Yaskawa INFORM job: X2_99(90,0).JBI

/JOB
//NAME X2_99(90,0)
///FOLDERNAME X2
//POS
///NPOS 429,429,425,13,0,0
///TOOL 0
///POSTYPE PULSE
///PULSE
C00000=-2065,-103387,-83817,35,52737,-27
C00001=166393,-132062,-92618,-58483,55149,-81008
C00002=157482,-99612,-82443,-50725,53832,76817
C00003=152781,-96239,-78741,-49340,50884,75750
C00004=150954,-94792,-77210,-48744,49760,75306
C00005=150957,-94045,-75225,-49281,49201,75681
C00006=151067,-94769,-77060,-48840,49767,75375
C00007=148896,-96259,-77631,-48213,48319,74911
C00008=154925,-106114,-81211,-52368,49780,77962
C00009=154976,-104737,-78409,-53070,49177,78455
C00010=153765,-101609,-77307,-52041,49068,77683
C00011=154727,-103781,-80113,-51957,49998,77663
C00012=157482,-99612,-82443,-50725,53832,76817
C00013=126812,-81448,-90767,-9472,77282,14340
C00014=120783,-85892,-98127,47,82159,-60
C00015=120791,-78998,-92147,45,82022,-58
C00016=120812,-59041,-81112,38,85486,-50
C00017=120812,-59638,-79752,38,84341,-50
C00018=120812,-59041,-81112,38,85486,-50
C00019=120792,-70899,-87175,45,83124,-57
C00020=120810,-72484,-85548,40,81307,-51
C00021=120817,-76009,-87202,37,80512,-50
C00022=120816,-72927,-85752,37,81205,-50
C00023=120792,-71723,-87920,45,83159,-57
C00024=120783,-85892,-98127,47,82159,-60
C00025=120841,-86418,-98444,30,82084,-41
C00026=120867,-62955,-84955,21,85839,-32
C00027=120862,-57449,-80347,23,85833,-34
C00028=120862,-58065,-78999,24,84687,-34
C00029=120862,-57449,-80347,23,85833,-34
C00030=120848,-76846,-90076,28,81853,-39
C00031=120700,-77430,-87681,72,80079,-89
C00032=120707,-73445,-85814,70,80978,-86
C00033=120700,-77430,-87681,72,80079,-89
C00034=120841,-86418,-98444,30,82084,-41
C00035=120877,-85820,-98106,19,82183,-30
C00036=120894,-60284,-82721,14,85837,-23
C00037=120891,-57831,-80469,15,85712,-24
C00038=120891,-58439,-79117,15,84567,-25
C00039=120891,-57831,-80469,15,85712,-24
C00040=120882,-76306,-89742,18,81925,-28
C00041=120632,-76849,-87581,92,80316,-111
C00042=120641,-72870,-85708,89,81208,-107
C00043=120899,-105607,-111704,13,80383,-24
C00044=120899,-105607,-111704,13,80383,-24
C00045=120329,-64675,-84682,181,84785,-205
C00046=120337,-61857,-81845,179,84488,-203
C00047=120337,-62228,-80870,179,83698,-204
C00048=120337,-61849,-81865,179,84506,-203
C00049=120308,-72964,-87409,188,82206,-216
C00050=112365,-66887,-81837,2540,82030,-2815
C00051=112466,-65041,-80903,2509,82400,-2777
C00052=112291,-68228,-82506,2565,81755,-2847
C00053=88690,-37051,-64863,22386,100281,-29037
C00054=90338,-32373,-60570,22143,99643,-28585
C00055=86677,-30127,-56933,28301,101078,-28609
C00056=87262,-30704,-57322,28229,100840,-28451
C00057=86036,-30845,-57417,28365,101220,-28810
C00058=80749,-50154,-73696,28906,103010,-30322
C00059=106026,-92840,-102541,4408,81700,-4909
C00060=104933,-21068,-63327,14588,98299,-15445
C00061=118026,-7058,-59426,-2478,121298,-42537
C00062=119206,-9959,-57512,-2402,118662,-42076
C00063=119679,-11008,-56668,-2374,117617,-41892
C00064=119678,-12040,-55711,-2348,116499,-41868
C00065=119679,-11008,-56668,-2374,117617,-41892
C00066=117888,-11929,-55575,-2351,116426,-42475
C00067=118578,-11982,-55616,-2350,116441,-42241
C00068=117888,-11929,-55575,-2351,116426,-42475
C00069=116239,-8118,-58416,-2447,120087,-43116
C00070=117941,-7017,-59404,-2478,121303,-42566
C00071=119121,-9922,-57492,-2402,118667,-42105
C00072=119594,-10972,-56650,-2375,117622,-41921
C00073=119593,-12004,-55694,-2348,116504,-41897
C00074=119594,-10972,-56650,-2375,117622,-41921
C00075=117972,-11968,-55595,-2351,116420,-42446
C00076=118663,-12020,-55635,-2349,116436,-42212
C00077=117972,-11968,-55595,-2351,116420,-42446
C00078=116323,-8162,-58441,-2447,120082,-43087
C00079=118213,-4464,-57342,-2479,121353,-42475
C00080=119375,-7335,-55445,-2404,118742,-42020
C00081=119840,-8375,-54609,-2376,117706,-41839
C00082=119839,-9401,-53662,-2350,116597,-41815
C00083=119840,-8375,-54609,-2376,117706,-41839
C00084=117787,-9255,-53494,-2353,116516,-42511
C00085=118466,-9310,-53537,-2352,116532,-42281
C00086=117787,-9255,-53494,-2353,116516,-42511
C00087=113921,-56504,-90793,659,90254,-43086
C00088=172997,-84117,-74043,-29270,60841,-12459
C00089=182497,-62439,-47217,-33561,35566,-5540
C00090=159932,16406,-23252,-17890,77970,-26070
C00091=160037,20332,-16581,-18068,76003,-25738
C00092=160078,21964,-13839,-18147,75202,-25602
C00093=160081,21492,-12606,-18227,74248,-25457
C00094=160088,21570,-12789,-18218,74396,-25476
C00095=160141,24413,-10063,-18259,74201,-25427
C00096=160088,21570,-12789,-18218,74396,-25476
C00097=159942,15886,-22293,-17945,77154,-25943
C00098=147845,25725,-14551,-15841,76328,-30554
C00099=147785,29164,-8153,-15217,74000,-30118
C00100=146391,29253,-6691,-12120,72163,-29888
C00101=146393,28810,-5449,-12184,71193,-29788
C00102=146383,28918,-5675,-12167,71382,-29809
C00103=146621,31717,-2885,-12295,71143,-29703
C00104=146383,28918,-5675,-12167,71382,-29809
C00105=147481,21483,-15847,-15359,72675,-30094
C00106=159281,-34086,-66545,-16207,79188,-23357
C00107=99248,-110920,-110752,20005,76383,-39509
C00108=66302,7791,-36486,37409,101463,8597
C00109=118447,29266,3056,46998,72230,30227
C00110=127168,50798,26938,44779,68662,26958
C00111=126741,52789,31626,47411,67245,26245
C00112=126739,52962,33479,47729,66520,25863
C00113=126722,52773,32881,47650,66716,25957
C00114=127164,55780,36224,47676,66131,25882
C00115=126722,52773,32881,47650,66716,25957
C00116=126349,45711,19766,44599,70372,27360
C00117=120505,26515,5919,45760,54508,48320
C00118=117448,33812,16008,47845,44948,58363
C00119=118470,38735,23995,49076,42786,57538
C00120=118868,40836,27368,49664,41907,57166
C00121=118868,41209,29429,50591,41201,56605
C00122=118874,41229,29076,50388,41345,56729
C00123=119426,43973,31977,50392,40796,56713
C00124=118874,41229,29076,50388,41345,56729
C00125=113429,42926,32106,63659,45667,52339
C00126=114748,48529,40817,65458,43685,51182
C00127=114893,50540,41231,64669,43936,51674
C00128=112305,42308,35228,66023,45399,50822
C00129=115273,50693,44169,66217,42928,50725
C00130=115426,53095,46610,68400,49137,42398
C00131=119344,57393,45281,61419,62909,27573
C00132=122643,57481,41003,55027,68134,22006
C00133=122245,55189,37420,54802,68977,22330
C00134=121107,49775,28783,54366,71151,23084
C00135=66302,7791,-36486,37409,101463,8597
C00136=87180,-51399,-85456,25144,96058,-16686
C00137=99248,-110920,-110752,20005,76383,-39509
C00138=111751,-62315,-95524,15437,88724,-33512
C00139=159281,-34086,-66545,-16207,79188,-23357
C00140=168180,19564,-18932,-27022,75314,-21681
C00141=167557,25730,-9148,-27095,72571,-21254
C00142=169085,37421,-2781,-29202,81184,-22287
C00143=169685,28444,-11845,-29359,82224,-22336
C00144=167557,25730,-9148,-27095,72571,-21254
C00145=149649,39094,-686,-15861,76123,-27675
C00146=150907,26639,-9385,-19166,68714,-26529
C00147=150787,22066,-16509,-18873,70615,-26886
C00148=159281,-34086,-66545,-16207,79188,-23357
C00149=152303,-102933,-107906,365,71882,-21471
C00150=121799,-34443,-59064,1710,93632,-36707
C00151=118945,163,-15392,1659,93503,-40633
C00152=120696,28796,14633,1549,89703,-40093
C00153=120597,41866,29081,1551,94027,-40072
C00154=120652,45714,33392,1563,96828,-40019
C00155=120580,21627,9250,1574,100354,-40001
C00156=120617,1336,-9032,1541,99246,-41820
C00157=120512,926,-9516,1535,99334,-41857
C00158=120163,-1908,-13337,1516,100237,-41964
C00159=118931,-1420,-16721,1449,102592,-42361
C00160=118945,163,-15392,1659,93503,-40633
C00161=120171,930,-10959,1582,91145,-40250
C00162=120660,1326,-9108,1553,90200,-40098
C00163=120694,25865,13192,1550,89085,-40100
C00164=120696,29026,16285,1550,88805,-40104
C00165=120258,23290,9189,1576,90234,-40233
C00166=119165,22386,4533,1644,92655,-40570
C00167=119181,24192,6266,1459,101602,-42286
C00168=120260,23811,9690,1517,99280,-41943
C00169=120693,23749,11149,1541,98342,-41806
C00170=120660,1326,-9108,1544,99287,-41805
C00171=120174,1432,-10536,1517,100229,-41961
C00172=118965,1918,-13913,1451,102579,-42349
C00173=119164,21752,3941,1459,101779,-42290
C00174=120255,21351,7351,1518,99456,-41942
C00175=120694,21281,8802,1542,98518,-41803
C00176=120641,1282,-9371,1543,99426,-41811
C00177=120163,-1908,-13337,1516,100237,-41964
C00178=118931,-1420,-16721,1449,102592,-42361
C00179=109578,15420,-7310,28367,110236,41857
C00180=109763,14188,-4345,27924,107995,41350
C00181=110205,13439,-3187,27787,106873,41241
C00182=131058,12711,-3863,29133,99851,47652
C00183=122151,9951,8068,53530,92588,44188
C00184=120623,10562,7326,53535,93941,44154
C00185=119164,10594,3761,53715,96134,44669
C00186=115308,-32515,-29810,53374,97452,43308
C00187=161838,-55085,-61541,-4908,86946,11244
C00188=151264,19092,-3987,-26397,112513,-34927
C00189=144058,12336,-10204,-27380,110553,-37342
C00190=143876,11528,-6807,-26938,108253,-36840
C00191=143883,12398,-4144,-26739,107186,-36580
C00192=138876,8905,-7310,-27290,105714,-38195
C00193=141808,11001,6672,-48404,103196,-38053
C00194=146391,20880,29557,-62395,105787,-26226
C00195=143524,10867,7651,-51737,104094,-37857
C00196=145724,13401,6310,-52003,106686,-38162
C00197=151264,19092,-3987,-26397,112513,-34927
C00198=161838,-55085,-61541,-4908,86946,11244
C00199=148116,-52831,-56464,-50581,83749,-77178
C00200=143654,-45216,-49088,-49944,80892,-77944
C00201=142056,-46762,-48840,-49795,79395,-77968
C00202=142218,-45304,-47887,-49802,79593,-77989
C00203=141353,-40392,-44909,-49565,79578,-78427
C00204=143095,-64861,-43193,-72743,55101,-56913
C00205=145645,-63649,-42384,-72835,56889,-56645
C00206=146567,-66336,-44709,-72863,57538,-56558
C00207=148638,-70217,-49243,-72528,59219,-56701
C00208=152439,-71702,-66380,-51300,83828,-74957
C00209=84213,-62636,-84550,16381,94117,-81885
C00210=95245,-30826,-59151,14149,92862,-78402
C00211=97191,-43170,-61473,15355,82699,-78714
C00212=98481,-44184,-62246,14992,82421,-78309
C00213=94037,-41035,-61513,16198,84364,-79567
C00214=63521,1839,6360,71273,102323,-80160
C00215=65526,-1458,4791,71319,100695,-80245
C00216=65441,-828,6596,71139,100483,-80605
C00217=61873,133,7709,70638,102845,-81131
C00218=97631,-84017,-82277,6042,71977,-80454
C00219=97631,-84017,-82277,6042,71977,-13540
C00220=100992,-100869,-74320,15072,37892,-15545
C00221=103157,-95187,-70426,13089,38023,-14317
C00222=103157,-92961,-65713,13621,36312,-14617
C00223=97699,-120955,-80408,20799,32327,-18909
C00224=-2043,-48212,-53796,8,82315,-15
C00225=-2043,-48212,-53796,8,82315,-15
C00226=-2043,-48212,-53796,8,82315,-15
C00227=-2043,-48212,-53796,8,82315,-15
C00228=-2043,-48212,-53796,8,82315,-15
C00229=50156,-143124,-107249,60088,69694,-78596
C00230=70410,-104162,-83449,55661,60383,-81011
C00231=84923,-92751,-76765,50721,53081,-76684
C00232=86734,-91468,-75289,50215,51915,-76295
C00233=86736,-90744,-73307,50726,51361,-76670
C00234=86623,-91438,-75136,50303,51925,-76361
C00235=88689,-93063,-75778,49797,50498,-75974
C00236=86623,-91438,-75136,50303,51925,-76361
C00237=82499,-102310,-79219,53526,52313,-78845
C00238=82460,-100986,-76424,54186,51705,-79335
C00239=83746,-97994,-75341,53258,51491,-78599
C00240=82460,-100986,-76424,54186,51705,-79335
C00241=83820,-89231,-90898,31984,73153,-45470
C00242=103333,-81093,-95821,5106,83352,-5547
C00243=105734,-58391,-81894,4383,86302,-4664
C00244=106051,-55558,-79074,4290,86007,-4572
C00245=106052,-56155,-77720,4294,84870,-4611
C00246=106051,-55558,-79074,4290,86007,-4572
C00247=104417,-72181,-87594,4790,82806,-5215
C00248=104401,-72744,-85473,4810,81218,-5281
C00249=104801,-68935,-83629,4684,82015,-5119
C00250=104401,-72744,-85473,4810,81218,-5281
C00251=103333,-81093,-95821,5106,83352,-5547
C00252=121034,-86160,-98106,-184,81635,191
C00253=120937,-60313,-84022,-154,86250,153
C00254=120931,-57182,-80055,-152,85416,152
C00255=120931,-57770,-78693,-152,84276,154
C00256=120931,-57182,-80055,-152,85416,152
C00257=120995,-76536,-89732,-172,81427,178
C00258=121142,-77068,-87314,-217,79666,229
C00259=121124,-73096,-85459,-211,80565,222
C00260=121142,-77068,-87314,-217,79666,229
C00261=121096,-115670,-111851,-205,74930,222
C00262=121096,-115670,-111851,-205,74930,222
C00263=111920,-77360,-89293,2569,80863,-2809
C00264=113418,-69208,-82911,2118,81083,-2310
C00265=113298,-70113,-82134,2157,80142,-2365
C00266=113298,-69851,-83365,2151,81033,-2349
C00267=112830,-79068,-87705,2304,78982,-2541
C00268=118405,-74923,-83336,614,78322,-682
C00269=118432,-73250,-82545,605,78695,-671
C00270=118359,-77891,-84712,629,77644,-701
C00271=147649,-49700,-70143,-21952,96038,28312
C00272=144092,-44169,-65180,-21423,94945,27268
C00273=143301,-44665,-65479,-21298,94683,27039
C00274=145130,-43494,-64769,-21581,95292,27566
C00275=153783,-86392,-93366,-22522,93398,30972
C00276=150910,-93017,-97560,-17688,85250,21630
C00277=120908,-62091,-84868,-144,85857,144
C00278=120903,-58004,-80414,-143,85215,144
C00279=120903,-58580,-79044,-143,84076,145
C00280=120903,-58004,-80414,-143,85215,144
C00281=120961,-76486,-89626,-161,81387,167
C00282=121210,-76970,-87437,-238,79792,251
C00283=121190,-72994,-85579,-231,80691,243
C00284=121210,-76970,-87437,-238,79792,251
C00285=120997,-86105,-97999,-172,81597,178
C00286=122173,-44832,-80249,1138,103105,21360
C00287=123342,-6609,-59067,2432,120936,42504
C00288=122164,-9458,-57119,2365,118305,42047
C00289=121693,-10486,-56262,2341,117263,41864
C00290=121692,-11496,-55292,2315,116147,41841
C00291=121693,-10486,-56262,2341,117263,41864
C00292=123082,-11418,-55178,2309,116084,42311
C00293=122789,-11440,-55197,2311,116090,42211
C00294=123477,-11388,-55156,2308,116075,42444
C00295=125124,-7649,-58044,2392,119728,43080
C00296=123427,-6569,-59045,2432,120941,42533
C00297=122249,-10161,-56477,2346,117547,42058
C00298=121777,-10451,-56245,2341,117268,41893
C00299=121777,-11461,-55275,2315,116153,41870
C00300=121777,-10451,-56245,2341,117268,41893
C00301=123393,-11428,-55177,2309,116069,42415
C00302=122704,-11478,-55216,2311,116085,42182
C00303=123393,-11428,-55177,2309,116069,42415
C00304=123141,-2998,-56146,2434,120999,42438
C00305=121991,-6366,-54527,2366,118305,41988
C00306=121527,-6824,-53376,2344,117373,41811
C00307=121527,-7826,-52419,2319,116269,41787
C00308=121527,-6824,-53376,2344,117373,41811
C00309=123560,-7684,-52253,2311,116189,42474
C00310=122887,-7737,-52295,2313,116204,42247
C00311=123560,-7684,-52253,2311,116189,42474
C00312=125171,-3981,-55094,2393,119797,43097
C00313=101327,-45531,-60072,2075,102128,34667
C00314=89266,4396,-33928,11465,93507,29927
C00315=71071,57081,18578,22711,75509,22099
C00316=71211,62019,27131,22931,72950,21646
C00317=71266,64149,30755,23040,71886,21453
C00318=71267,63961,32200,23162,70975,21270
C00319=71260,64000,31991,23145,71114,21296
C00320=71334,67369,35901,23203,70471,21193
C00321=71260,64000,31991,23145,71114,21296
C00322=71066,56762,19636,22790,74756,21949
C00323=94467,40678,813,12417,73109,29814
C00324=94083,44902,8245,12754,70817,29441
C00325=93934,46692,11343,12898,69876,29287
C00326=93935,46363,12659,12975,68921,29182
C00327=93944,46449,12421,12955,69106,29206
C00328=93737,49413,15622,13089,68702,29088
C00329=93944,46449,12421,12955,69106,29206
C00330=94477,40302,1770,12461,72343,29738
C00331=89266,4396,-33928,11465,93507,29927
C00332=101327,-45531,-60072,2075,102128,34667
C00333=154347,-58865,-59313,-31959,84488,-20300
C00334=132804,-7309,-34611,-38234,83249,-26564
C00335=122176,70455,38125,-50476,77977,-25755
C00336=115295,79862,53015,-49496,71409,-25751
C00337=115674,81709,55615,-49754,71183,-25426
C00338=115674,81913,57390,-49999,70533,-25064
C00339=115723,81771,56361,-49871,70928,-25259
C00340=115127,86395,62081,-50016,69849,-24976
C00341=115723,81734,56059,-49831,71039,-25319
C00342=117859,70375,39301,-49439,75156,-26443
C00343=124576,6255,-12780,-47438,56902,-47453
C00344=122250,19334,1935,-46182,44641,-59320
C00345=122250,19334,1935,-46182,44641,-59320
C00346=120782,25934,12333,-47564,41782,-58376
C00347=120782,26215,14271,-48443,41066,-57848
C00348=120776,26249,13930,-48246,41217,-57966
C00349=120208,28831,16455,-48074,40759,-58046
C00350=120776,26249,13930,-48246,41217,-57966
C00351=118681,43368,36578,-62815,38306,-52785
C00352=118657,41916,32618,-60942,39123,-53866
C00353=119090,39280,31915,-62143,38937,-53171
C00354=118568,43405,36686,-62818,38211,-52783
C00355=112564,55763,35688,-55377,68087,-24843
C00356=113391,48910,28472,-52811,66916,-24378
C00357=112985,43681,22401,-52223,67232,-24845
C00358=132804,-7309,-34611,-38234,83249,-26564
C00359=154347,-58865,-59313,-31959,84488,-20300
C00360=101327,-45531,-60072,2075,102128,34667
C00361=89266,4396,-33928,11465,93507,29927
C00362=66565,54061,16600,30569,73521,18779
C00363=67024,59337,25188,30775,71132,18293
C00364=67157,61403,28617,30898,70179,18077
C00365=81564,59654,26436,24505,65914,22675
C00366=81641,57287,22841,24296,66807,22900
C00367=81527,51927,14208,23948,69183,23371
C00368=78027,-14448,-47618,10307,89336,23924
C00369=122403,540,-15029,-1679,93098,40614
C00370=116416,39963,24023,-1992,100377,38466
C00371=113398,50152,38563,-2230,96586,37494
C00372=112489,24468,12107,-2384,100085,37116
C00373=111594,3062,-7595,-2103,98667,38669
C00374=111355,667,-9500,-2114,98597,38588
C00375=111941,198,-11543,-2089,99632,38773
C00376=113186,289,-15256,-2035,101994,39161
C00377=122403,540,-15029,-1679,93098,40614
C00378=121179,1356,-10556,-1597,90741,40233
C00379=120574,1774,-8687,-1557,89793,40041
C00380=120532,26429,13697,-1554,88684,40039
C00381=121099,23723,9564,-1591,89850,40218
C00382=122190,22771,4863,-1663,92275,40553
C00383=122175,24579,6594,-1485,101224,42269
C00384=121098,24245,10065,-1538,98897,41927
C00385=120630,24202,11544,-1561,97957,41779
C00386=120666,1773,-8688,-1564,98883,41779
C00387=121177,1858,-10134,-1538,99825,41943
C00388=122384,2295,-13553,-1478,102176,42330
C00389=122189,22661,4761,-1485,101367,42272
C00390=121101,22312,8220,-1538,99039,41927
C00391=120664,22262,9692,-1560,98100,41789
C00392=120644,766,-9415,-1564,98810,41771
C00393=121185,-971,-12517,-1537,99838,41946
C00394=122412,-533,-15942,-1476,102193,42339
C00395=131781,15460,-7279,-28376,109886,-41795
C00396=131592,14275,-4268,-27940,107640,-41290
C00397=130646,14147,-2566,-27857,106338,-41338
C00398=110382,14201,-2350,-29042,99390,-47524
C00399=119227,11935,9973,-53508,92244,-44000
C00400=120732,10849,7590,-53521,93669,-44023
C00401=122191,10834,3980,-53696,95864,-44539
C00402=128646,-26020,-30624,-53883,101032,-13133
C00403=66557,-34885,-48546,20214,102394,2504
C00404=79484,36547,13079,24373,114005,30975
C00405=85904,26694,3247,25718,112997,33343
C00406=86041,25965,6661,25253,110710,32858
C00407=85714,26763,9282,24984,109715,32500
C00408=90422,20837,3523,25806,108738,34143
C00409=87739,24554,20424,48221,108657,34815
C00410=84755,20942,20954,53722,106133,35573
C00411=84755,20942,20954,53722,106133,35573
C00412=84776,24179,21069,50511,109377,34699
C00413=84698,26318,18454,50015,112057,35133
C00414=81578,31234,5255,15438,110633,30982
C00415=71416,-31459,-49219,37385,106309,54903
C00416=79334,-27512,-40554,52438,93314,75230
C00417=81671,-29746,-39165,52092,90747,74997
C00418=82501,-31675,-39268,51984,89697,74838
C00419=82828,-30755,-38544,51956,89529,74918
C00420=84142,-26044,-35343,51821,89078,75358
C00421=80223,-43644,-36659,65279,74230,62526
C00422=80042,-45349,-41066,60562,72331,65280
C00423=77493,-50941,-36554,72626,70323,55695
C00424=74018,-52299,-39928,72336,73171,55924
C00425=60945,-55409,-65093,53734,104166,71681
C00426=60945,-55409,-65093,53734,104166,71681
C00427=122092,-114409,-88723,-8345,70481,11232
C00428=-2000,-48025,-60869,0,102856,0
BC00000=781,523905,302382
BC00001=30742,515701,66855
BC00002=31638,515479,60490
BC00003=31638,515479,60490
BC00004=31638,515479,60490
BC00005=31638,515479,60490
BC00006=31638,515479,60490
BC00007=31638,515479,60490
BC00008=31638,515479,60490
BC00009=31638,515479,60490
BC00010=31638,515479,60490
BC00011=31638,515479,60490
BC00012=31638,515479,60490
BC00013=13239,522628,91328
BC00014=10409,517207,59294
BC00015=10409,517207,59294
BC00016=10409,517207,59294
BC00017=10409,517207,59294
BC00018=10409,517207,59294
BC00019=10409,517207,59294
BC00020=10409,517207,59294
BC00021=10409,517207,59294
BC00022=10409,517207,59294
BC00023=10409,517207,59294
BC00024=10409,517207,59294
BC00025=68218,516454,58706
BC00026=68218,516454,58706
BC00027=68218,516454,58706
BC00028=68218,516454,58706
BC00029=68218,516454,58706
BC00030=68218,516454,58706
BC00031=68218,516454,58706
BC00032=68218,516454,58706
BC00033=68218,516454,58706
BC00034=68218,516454,58706
BC00035=126843,516488,59263
BC00036=126843,516488,59263
BC00037=126843,516488,59263
BC00038=126843,516488,59263
BC00039=126843,516488,59263
BC00040=126843,516488,59263
BC00041=126843,516488,59263
BC00042=126843,516488,59263
BC00043=126843,520400,59263
BC00044=387083,520400,59263
BC00045=387083,520400,59263
BC00046=387083,520400,59263
BC00047=387083,520400,59263
BC00048=387083,520400,59263
BC00049=387083,520400,59263
BC00050=387083,520400,59263
BC00051=387083,520400,59263
BC00052=387083,520400,59263
BC00053=387083,520400,59263
BC00054=387083,520400,59263
BC00055=387083,520400,59263
BC00056=387083,520400,59263
BC00057=387083,520400,59263
BC00058=387083,520400,59263
BC00059=126843,518210,59263
BC00060=126843,518210,59263
BC00061=129574,490644,58205
BC00062=129574,490644,58205
BC00063=129574,490644,58205
BC00064=129574,490644,58205
BC00065=129574,490644,58205
BC00066=129574,490644,58205
BC00067=129574,490644,58205
BC00068=129574,490644,58205
BC00069=129574,490644,58205
BC00070=129597,444075,57932
BC00071=129597,444075,57932
BC00072=129597,444075,57932
BC00073=129597,444075,57932
BC00074=129597,444075,57932
BC00075=129597,444075,57932
BC00076=129597,444075,57932
BC00077=129597,444075,57932
BC00078=129597,444075,57932
BC00079=128889,400556,57777
BC00080=128889,400556,57777
BC00081=128889,400556,57777
BC00082=128889,400556,57777
BC00083=128889,400556,57777
BC00084=128889,400556,57777
BC00085=128889,400556,57777
BC00086=128889,400556,57777
BC00087=128889,400556,57777
BC00088=181249,400556,192761
BC00089=202914,400556,241573
BC00090=123650,400556,63155
BC00091=123650,400556,63155
BC00092=123650,400556,63155
BC00093=123650,400556,63155
BC00094=123650,400556,63155
BC00095=123650,400556,63155
BC00096=123650,400556,63155
BC00097=123650,400556,63155
BC00098=128418,400556,63301
BC00099=128418,400556,63301
BC00100=128418,400556,63301
BC00101=128418,400556,63301
BC00102=128418,400556,63301
BC00103=128418,400556,63301
BC00104=128418,400556,63301
BC00105=128418,400556,63301
BC00106=120912,400556,90455
BC00107=91224,400556,32086
BC00108=60523,400556,81483
BC00109=120036,400556,87759
BC00110=141181,415917,88489
BC00111=141181,415917,88489
BC00112=141181,415917,88489
BC00113=141181,415917,88489
BC00114=141181,415917,88489
BC00115=141181,415917,88489
BC00116=141181,415917,88489
BC00117=135777,415917,84971
BC00118=132933,415917,83120
BC00119=132933,415917,83120
BC00120=132933,415917,83120
BC00121=132933,415917,83120
BC00122=132933,415917,83120
BC00123=132933,415917,83120
BC00124=132933,415917,83120
BC00125=133247,415917,81483
BC00126=133247,415917,81483
BC00127=133247,415917,81483
BC00128=133247,415917,81483
BC00129=133246,415917,81483
BC00130=133247,415917,81482
BC00131=133247,415917,81483
BC00132=133247,415917,81483
BC00133=133247,415917,81483
BC00134=133247,415917,81483
BC00135=60523,400556,81483
BC00136=78278,400556,52915
BC00137=91224,400556,32086
BC00138=91224,400556,32086
BC00139=120912,400556,90455
BC00140=136017,400556,32086
BC00141=136017,400556,32086
BC00142=136017,400556,32086
BC00143=136017,400556,32086
BC00144=136017,400556,32086
BC00145=136017,400556,32086
BC00146=136017,400556,32086
BC00147=136017,400556,32086
BC00148=120912,400556,90455
BC00149=158121,400556,32086
BC00150=123507,424612,191697
BC00151=141020,441223,281235
BC00152=141020,441223,281235
BC00153=141020,441223,281235
BC00154=141020,441223,281235
BC00155=141020,441223,281235
BC00156=141154,470147,281572
BC00157=141330,514662,281853
BC00158=141330,514662,281853
BC00159=141330,514662,281853
BC00160=143409,441223,281235
BC00161=143409,441223,281235
BC00162=143409,441223,281235
BC00163=143409,441223,281235
BC00164=143409,441223,281235
BC00165=143409,441223,281235
BC00166=143409,441223,281235
BC00167=143543,470147,281572
BC00168=143543,470147,281572
BC00169=143543,470147,281572
BC00170=143543,470147,281572
BC00171=143543,470147,281572
BC00172=143543,470147,281572
BC00173=143719,514662,281853
BC00174=143719,514662,281853
BC00175=143719,514662,281853
BC00176=143719,514662,281853
BC00177=143719,514662,281853
BC00178=143719,514662,281853
BC00179=144290,523889,221847
BC00180=144290,523889,221847
BC00181=144290,523889,221847
BC00182=144290,523889,221847
BC00183=144290,523889,221845
BC00184=144290,523889,221847
BC00185=144290,523889,221847
BC00186=144290,523889,221847
BC00187=796,523889,224399
BC00188=796,523889,224399
BC00189=796,523889,224399
BC00190=796,523889,224399
BC00191=796,523889,224399
BC00192=796,523889,224399
BC00193=796,523889,224399
BC00194=796,523889,224399
BC00195=796,523889,224399
BC00196=796,523889,224399
BC00197=796,523889,224399
BC00198=796,523889,224399
BC00199=797,523888,121430
BC00200=796,523889,121434
BC00201=796,523889,121434
BC00202=796,523889,121434
BC00203=796,523889,121434
BC00204=796,523889,121434
BC00205=796,523889,121434
BC00206=796,523889,121434
BC00207=796,523889,121434
BC00208=796,523889,121434
BC00209=380682,523889,121434
BC00210=380682,523889,121434
BC00211=380682,523889,121434
BC00212=380682,523889,121434
BC00213=380682,523889,121434
BC00214=380682,523889,121434
BC00215=380682,523889,121434
BC00216=380682,523889,121434
BC00217=380682,523889,121434
BC00218=380682,523889,121434
BC00219=380682,523889,121434
BC00220=380682,523889,121434
BC00221=380682,523889,121434
BC00222=380682,523889,121434
BC00223=380682,523889,121434
BC00224=796,523889,1075193
BC00225=796,523889,1075193
BC00226=796,523889,1075193
BC00227=796,523889,1075193
BC00228=796,584159,1075193
BC00229=395769,514369,57931
BC00230=395769,514369,57931
BC00231=395769,514369,57931
BC00232=395769,514369,57931
BC00233=395769,514369,57931
BC00234=395769,514369,57931
BC00235=395769,514369,57931
BC00236=395769,514369,57931
BC00237=395769,514369,57931
BC00238=395769,514369,57931
BC00239=395769,514369,57931
BC00240=395769,514369,57931
BC00241=395769,515177,57354
BC00242=395769,516086,56705
BC00243=395769,516086,56705
BC00244=395769,516086,56705
BC00245=395769,516086,56705
BC00246=395769,516086,56705
BC00247=395769,516086,56705
BC00248=395769,516086,56705
BC00249=395769,516086,56705
BC00250=395769,516086,56705
BC00251=395769,516086,56705
BC00252=364519,515355,56108
BC00253=364519,515355,56108
BC00254=364519,515355,56108
BC00255=364519,515355,56108
BC00256=364519,515355,56108
BC00257=364519,515355,56108
BC00258=364519,515355,56108
BC00259=364519,515355,56108
BC00260=364519,515355,56108
BC00261=364519,515355,56108
BC00262=28307,515355,56108
BC00263=28307,516891,68607
BC00264=28307,516891,73984
BC00265=28307,516891,73984
BC00266=28307,516891,73984
BC00267=28307,516891,73984
BC00268=28307,516891,73984
BC00269=28307,516891,73984
BC00270=28307,516891,73984
BC00271=28307,516891,73984
BC00272=28307,516891,73984
BC00273=28307,516891,73984
BC00274=28307,516891,73984
BC00275=28307,516891,73984
BC00276=336711,509467,91104
BC00277=305893,515413,56636
BC00278=305893,515413,56636
BC00279=305893,515413,56636
BC00280=305893,515413,56636
BC00281=305893,515413,56636
BC00282=305893,515413,56636
BC00283=305893,515413,56636
BC00284=305893,515413,56636
BC00285=305893,515413,56636
BC00286=304523,502491,56408
BC00287=303152,489569,56181
BC00288=303152,489569,56181
BC00289=303152,489569,56181
BC00290=303152,489569,56181
BC00291=303152,489569,56181
BC00292=303152,489569,56181
BC00293=303152,489569,56181
BC00294=303152,489569,56181
BC00295=303152,489569,56181
BC00296=303109,443000,56994
BC00297=303109,443000,56994
BC00298=303109,443000,56994
BC00299=303109,443000,56994
BC00300=303109,443000,56994
BC00301=303109,443000,56994
BC00302=303109,443000,56994
BC00303=303109,443000,56994
BC00304=303797,400556,57919
BC00305=303797,400556,57919
BC00306=303797,400556,57919
BC00307=303797,400556,57919
BC00308=303797,400556,57919
BC00309=303797,400556,57919
BC00310=303797,400556,57919
BC00311=303797,400556,57919
BC00312=303797,400556,57919
BC00313=303797,400556,221955
BC00314=296099,410471,136295
BC00315=257856,418698,65216
BC00316=257856,418698,65216
BC00317=257856,418698,65216
BC00318=257856,418698,65216
BC00319=257856,418698,65216
BC00320=257856,418698,65216
BC00321=257856,418698,65216
BC00322=257856,418698,65216
BC00323=294733,415445,65881
BC00324=294733,415445,65881
BC00325=294733,415445,65881
BC00326=294733,415445,65881
BC00327=294733,415445,65881
BC00328=294733,415445,65881
BC00329=294733,415445,65881
BC00330=294733,415445,65881
BC00331=296099,410471,136295
BC00332=303797,400556,221955
BC00333=303797,400556,221955
BC00334=298676,400556,147304
BC00335=307528,431278,26398
BC00336=283636,431278,26398
BC00337=283636,431278,26398
BC00338=283636,431278,26398
BC00339=283636,431278,26398
BC00340=283636,431278,26398
BC00341=283636,431278,26398
BC00342=283636,431278,26398
BC00343=294823,400556,85625
BC00344=294931,400556,84298
BC00345=294931,400556,84298
BC00346=294931,400556,84298
BC00347=294931,400556,84298
BC00348=294931,400556,84298
BC00349=294931,400556,84298
BC00350=294931,400556,84298
BC00351=276015,408236,82027
BC00352=276015,408236,82027
BC00353=276015,408236,82027
BC00354=276015,408236,82027
BC00355=275463,408352,55361
BC00356=276012,408236,82027
BC00357=276015,408236,82027
BC00358=298676,400556,147304
BC00359=303797,400556,221955
BC00360=303797,400556,221955
BC00361=296099,410471,136295
BC00362=257149,416120,34454
BC00363=257149,416120,34454
BC00364=257149,416120,34454
BC00365=257149,416120,34454
BC00366=257149,416120,34454
BC00367=257149,416120,34454
BC00368=262502,428258,159266
BC00369=291631,440131,281365
BC00370=278652,440131,281365
BC00371=267739,440131,281365
BC00372=267739,440131,281365
BC00373=267671,469055,280615
BC00374=267515,514115,279786
BC00375=267515,514115,279786
BC00376=267515,514115,279786
BC00377=294020,440131,281365
BC00378=294020,440131,281365
BC00379=294020,440131,281365
BC00380=294020,440131,281365
BC00381=294020,440131,281365
BC00382=294020,440131,281365
BC00383=293952,469055,280615
BC00384=293952,469055,280615
BC00385=293952,469055,280615
BC00386=293952,469055,280615
BC00387=293952,469055,280615
BC00388=293952,469055,280615
BC00389=293796,514115,279786
BC00390=293796,514115,279786
BC00391=293796,514115,279786
BC00392=293796,514115,279786
BC00393=293796,514115,279786
BC00394=293796,514115,279786
BC00395=288422,523889,220135
BC00396=288422,523889,220135
BC00397=288422,523889,220135
BC00398=288422,523889,220135
BC00399=288422,523889,220135
BC00400=288422,523889,220135
BC00401=288422,523889,220135
BC00402=288422,523889,220135
BC00403=395769,523889,222081
BC00404=395769,523889,222081
BC00405=395769,523889,222081
BC00406=395769,523889,222081
BC00407=395769,523889,222081
BC00408=395769,523889,222081
BC00409=395769,523889,222080
BC00410=395769,523889,222080
BC00411=395769,523889,222080
BC00412=395769,523889,222081
BC00413=395769,523889,222081
BC00414=395769,523889,222081
BC00415=395769,523889,160664
BC00416=395769,523889,116189
BC00417=395769,523889,116189
BC00418=395769,523889,116189
BC00419=395769,523889,116189
BC00420=395769,523889,116189
BC00421=395769,523889,116189
BC00422=395769,523889,116189
BC00423=395769,523889,116189
BC00424=395769,523889,116189
BC00425=395769,523889,116189
BC00426=56749,523889,116189
BC00427=63741,523891,182530
BC00428=116059,523905,678960
EC00000=-798156,-183832
EC00001=-798156,-183832
EC00002=-798156,-183832
EC00003=-798156,-183832
EC00004=-798156,-183832
EC00005=-798156,-183832
EC00006=-798156,-183832
EC00007=-798156,-183832
EC00008=-798156,-183832
EC00009=-798156,-183832
EC00010=-798156,-183832
EC00011=-798156,-183832
EC00012=-798156,-183832
EC00013=-798156,-183832
EC00014=-798156,-183832
EC00015=-798156,-183832
EC00016=-798156,-183832
EC00017=-798156,-183832
EC00018=-798156,-183832
EC00019=-798156,-183832
EC00020=-798156,-183832
EC00021=-798156,-183832
EC00022=-798156,-183832
EC00023=-798156,-183832
EC00024=-798156,-183832
EC00025=-798156,-183832
EC00026=-798156,-183832
EC00027=-798156,-183832
EC00028=-798156,-183832
EC00029=-798156,-183832
EC00030=-798156,-183832
EC00031=-798156,-183832
EC00032=-798156,-183832
EC00033=-798156,-183832
EC00034=-798156,-183832
EC00035=-798156,-183832
EC00036=-798156,-183832
EC00037=-798156,-183832
EC00038=-798156,-183832
EC00039=-798156,-183832
EC00040=-798156,-183832
EC00041=-798156,-183832
EC00042=-798156,-183832
EC00043=-798156,-183832
EC00044=-798156,-183832
EC00045=-798156,-183832
EC00046=-798156,-183832
EC00047=-798156,-183832
EC00048=-798156,-183832
EC00049=-798156,-183832
EC00050=-798156,-183832
EC00051=-798156,-183832
EC00052=-798156,-183832
EC00053=-798156,-183832
EC00054=-798156,-183832
EC00055=-798156,-183832
EC00056=-798156,-183832
EC00057=-798156,-183832
EC00058=-798156,-183832
EC00059=-798156,-183832
EC00060=-798156,-183832
EC00061=-798156,-183832
EC00062=-798156,-183832
EC00063=-798156,-183832
EC00064=-798156,-183832
EC00065=-798156,-183832
EC00066=-798156,-183832
EC00067=-798156,-183832
EC00068=-798156,-183832
EC00069=-798156,-183832
EC00070=-798156,-183832
EC00071=-798156,-183832
EC00072=-798156,-183832
EC00073=-798156,-183832
EC00074=-798156,-183832
EC00075=-798156,-183832
EC00076=-798156,-183832
EC00077=-798156,-183832
EC00078=-798156,-183832
EC00079=-798156,-183832
EC00080=-798156,-183832
EC00081=-798156,-183832
EC00082=-798156,-183832
EC00083=-798156,-183832
EC00084=-798156,-183832
EC00085=-798156,-183832
EC00086=-798156,-183832
EC00087=-798156,-183832
EC00088=-798156,-183832
EC00089=-798156,-183832
EC00090=-798156,-183832
EC00091=-798156,-183832
EC00092=-798156,-183832
EC00093=-798156,-183832
EC00094=-798156,-183832
EC00095=-798156,-183832
EC00096=-798156,-183832
EC00097=-798156,-183832
EC00098=-798156,-183832
EC00099=-798156,-183832
EC00100=-798156,-183832
EC00101=-798156,-183832
EC00102=-798156,-183832
EC00103=-798156,-183832
EC00104=-798156,-183832
EC00105=-798156,-183832
EC00106=-798156,-183832
EC00107=-798156,-183832
EC00108=-798156,-183832
EC00109=-798156,-183832
EC00110=-798156,-183832
EC00111=-798156,-183832
EC00112=-798156,-183832
EC00113=-798156,-183832
EC00114=-798156,-183832
EC00115=-798156,-183832
EC00116=-798156,-183832
EC00117=-798156,-183832
EC00118=-798156,-183832
EC00119=-798156,-183832
EC00120=-798156,-183832
EC00121=-798156,-183832
EC00122=-798156,-183832
EC00123=-798156,-183832
EC00124=-798156,-183832
EC00125=-798156,-183832
EC00126=-798156,-183832
EC00127=-798155,-183833
EC00128=-798155,-183833
EC00129=-798156,-183832
EC00130=-798156,-183832
EC00131=-798156,-183832
EC00132=-798156,-183832
EC00133=-798156,-183832
EC00134=-798156,-183832
EC00135=-798156,-183832
EC00136=-798156,-183832
EC00137=-798156,-183832
EC00138=-798156,-183832
EC00139=-798156,-183832
EC00140=-798156,-183832
EC00141=-798156,-183832
EC00142=-798156,-183832
EC00143=-798156,-183832
EC00144=-798156,-183832
EC00145=-798156,-183832
EC00146=-798156,-183832
EC00147=-798156,-183832
EC00148=-798156,-183832
EC00149=-798156,-183832
EC00150=-798156,-183832
EC00151=-798156,-183832
EC00152=-798156,-183832
EC00153=-798156,-183832
EC00154=-798156,-183832
EC00155=-798156,-183832
EC00156=-798156,-183832
EC00157=-798156,-183832
EC00158=-798156,-183832
EC00159=-798156,-183832
EC00160=-798156,-183832
EC00161=-798156,-183832
EC00162=-798156,-183832
EC00163=-798156,-183832
EC00164=-798156,-183832
EC00165=-798156,-183832
EC00166=-798156,-183832
EC00167=-798156,-183832
EC00168=-798156,-183832
EC00169=-798156,-183832
EC00170=-798156,-183832
EC00171=-798156,-183832
EC00172=-798156,-183832
EC00173=-798156,-183832
EC00174=-798156,-183832
EC00175=-798156,-183832
EC00176=-798156,-183832
EC00177=-798156,-183832
EC00178=-798156,-183832
EC00179=-798155,-183833
EC00180=-798156,-183832
EC00181=-798156,-183832
EC00182=-798156,-183832
EC00183=-798156,-183832
EC00184=-798156,-183832
EC00185=-798156,-183832
EC00186=-798156,-183832
EC00187=-798156,-183832
EC00188=-798156,-183832
EC00189=-798156,-183832
EC00190=-798156,-183832
EC00191=-798156,-183832
EC00192=-798156,-183832
EC00193=-798156,-183832
EC00194=-798156,-183832
EC00195=-798155,-183832
EC00196=-798156,-183832
EC00197=-798156,-183832
EC00198=-798156,-183832
EC00199=-798156,-183832
EC00200=-798156,-183832
EC00201=-798156,-183832
EC00202=-798156,-183832
EC00203=-798156,-183832
EC00204=-798156,-183832
EC00205=-798156,-183832
EC00206=-798156,-183832
EC00207=-798156,-183832
EC00208=-798156,-183832
EC00209=-798156,-183832
EC00210=-798156,-183832
EC00211=-798156,-183832
EC00212=-798156,-183832
EC00213=-798156,-183832
EC00214=-798156,-183832
EC00215=-798156,-183832
EC00216=-798156,-183832
EC00217=-798156,-183832
EC00218=-798156,-183832
EC00219=-798156,-183832
EC00220=-798156,-183832
EC00221=-310394,-183832
EC00222=-310394,-740307
EC00223=-310394,-1296783
EC00224=-798156,-1296783
EC00225=-798156,-1296783
EC00226=-798156,-1296783
EC00227=-798156,-1296783
EC00228=-798156,-1296783
EC00229=-798156,-1296783
EC00230=-798156,-1296783
EC00231=-798156,-1296783
EC00232=-798156,-1296783
EC00233=-798156,-1296783
EC00234=-798156,-1296783
EC00235=-798156,-1296783
EC00236=-798156,-1296783
EC00237=-798156,-1296783
EC00238=-798156,-1296783
EC00239=-798156,-1296783
EC00240=-798156,-1296783
EC00241=-798156,-1296783
EC00242=-798156,-1296783
EC00243=-798156,-1296783
EC00244=-798156,-1296783
EC00245=-798156,-1296783
EC00246=-798156,-1296783
EC00247=-798156,-1296783
EC00248=-798156,-1296783
EC00249=-798156,-1296783
EC00250=-798156,-1296783
EC00251=-798156,-1296783
EC00252=-798156,-1296783
EC00253=-798156,-1296783
EC00254=-798156,-1296783
EC00255=-798156,-1296783
EC00256=-798156,-1296783
EC00257=-798156,-1296783
EC00258=-798156,-1296783
EC00259=-798156,-1296783
EC00260=-798156,-1296783
EC00261=-798156,-1296783
EC00262=-798156,-1296783
EC00263=-798156,-1296783
EC00264=-798156,-1296783
EC00265=-798156,-1296783
EC00266=-798156,-1296783
EC00267=-798156,-1296783
EC00268=-798156,-1296783
EC00269=-798156,-1296783
EC00270=-798156,-1296783
EC00271=-798156,-1296783
EC00272=-798156,-1296783
EC00273=-798156,-1296783
EC00274=-798156,-1296783
EC00275=-798156,-1296783
EC00276=-798156,-1296783
EC00277=-798156,-1296783
EC00278=-798156,-1296783
EC00279=-798156,-1296783
EC00280=-798156,-1296783
EC00281=-798156,-1296783
EC00282=-798156,-1296783
EC00283=-798156,-1296783
EC00284=-798156,-1296783
EC00285=-798156,-1296783
EC00286=-798156,-1296783
EC00287=-798156,-1296783
EC00288=-798156,-1296783
EC00289=-798156,-1296783
EC00290=-798156,-1296783
EC00291=-798156,-1296783
EC00292=-798156,-1296783
EC00293=-798156,-1296783
EC00294=-798156,-1296783
EC00295=-798156,-1296783
EC00296=-798156,-1296783
EC00297=-798156,-1296783
EC00298=-798156,-1296783
EC00299=-798156,-1296783
EC00300=-798156,-1296783
EC00301=-798156,-1296783
EC00302=-798156,-1296783
EC00303=-798156,-1296783
EC00304=-798156,-1296783
EC00305=-798156,-1296783
EC00306=-798156,-1296783
EC00307=-798156,-1296783
EC00308=-798156,-1296783
EC00309=-798156,-1296783
EC00310=-798156,-1296783
EC00311=-798156,-1296783
EC00312=-798156,-1296783
EC00313=-798156,-1296783
EC00314=-798156,-1296783
EC00315=-798156,-1296783
EC00316=-798156,-1296783
EC00317=-798156,-1296783
EC00318=-798156,-1296783
EC00319=-798156,-1296783
EC00320=-798156,-1296783
EC00321=-798156,-1296783
EC00322=-798156,-1296783
EC00323=-798156,-1296783
EC00324=-798156,-1296783
EC00325=-798156,-1296783
EC00326=-798156,-1296783
EC00327=-798156,-1296783
EC00328=-798156,-1296783
EC00329=-798156,-1296783
EC00330=-798156,-1296783
EC00331=-798156,-1296783
EC00332=-798156,-1296783
EC00333=-798156,-1296783
EC00334=-798156,-1296783
EC00335=-798156,-1296783
EC00336=-798156,-1296783
EC00337=-798156,-1296783
EC00338=-798156,-1296783
EC00339=-798156,-1296783
EC00340=-798156,-1296783
EC00341=-798156,-1296783
EC00342=-798156,-1296783
EC00343=-798156,-1296783
EC00344=-798156,-1296783
EC00345=-798156,-1296783
EC00346=-798156,-1296783
EC00347=-798156,-1296783
EC00348=-798156,-1296783
EC00349=-798156,-1296783
EC00350=-798156,-1296783
EC00351=-798156,-1296783
EC00352=-798156,-1296783
EC00353=-798156,-1296783
EC00354=-798156,-1296783
EC00355=-798156,-1296783
EC00356=-798156,-1296783
EC00357=-798156,-1296783
EC00358=-798156,-1296783
EC00359=-798156,-1296783
EC00360=-798156,-1296783
EC00361=-798156,-1296783
EC00362=-798156,-1296783
EC00363=-798156,-1296783
EC00364=-798156,-1296783
EC00365=-798156,-1296783
EC00366=-798156,-1296783
EC00367=-798156,-1296783
EC00368=-798156,-1296783
EC00369=-798156,-1296783
EC00370=-798156,-1296783
EC00371=-798156,-1296783
EC00372=-798156,-1296783
EC00373=-798156,-1296783
EC00374=-798156,-1296783
EC00375=-798156,-1296783
EC00376=-798156,-1296783
EC00377=-798156,-1296783
EC00378=-798156,-1296783
EC00379=-798156,-1296783
EC00380=-798156,-1296783
EC00381=-798156,-1296783
EC00382=-798156,-1296783
EC00383=-798156,-1296783
EC00384=-798156,-1296783
EC00385=-798156,-1296783
EC00386=-798156,-1296783
EC00387=-798156,-1296783
EC00388=-798156,-1296783
EC00389=-798156,-1296783
EC00390=-798156,-1296783
EC00391=-798156,-1296783
EC00392=-798156,-1296783
EC00393=-798156,-1296783
EC00394=-798156,-1296783
EC00395=-798156,-1296783
EC00396=-798156,-1296783
EC00397=-798156,-1296783
EC00398=-798156,-1296783
EC00399=-798156,-1296783
EC00400=-798156,-1296783
EC00401=-798156,-1296783
EC00402=-798156,-1296783
EC00403=-798156,-1296783
EC00404=-798156,-1296783
EC00405=-798154,-1296781
EC00406=-798154,-1296781
EC00407=-798154,-1296781
EC00408=-798155,-1296782
EC00409=-798156,-1296783
EC00410=-798156,-1296783
EC00411=-798156,-1296783
EC00412=-798156,-1296783
EC00413=-798156,-1296783
EC00414=-798156,-1296783
EC00415=-798156,-1296783
EC00416=-798156,-1296783
EC00417=-798156,-1296783
EC00418=-798156,-1296783
EC00419=-798156,-1296783
EC00420=-798156,-1296783
EC00421=-798156,-1296783
EC00422=-798156,-1296783
EC00423=-798154,-1296780
EC00424=-798156,-1296783
///POSTYPE BASE
///RECTAN
///RCONF 0,0,0,0,1,0,0,0,0,0,0,0,0,0,0,0,0,0,0,0,0,0,0,0
P00006=2.006,1.622,-0.565,0.0000,0.0000,0.0000
P00021=0.073,2.058,-0.109,0.0000,0.0000,0.0000
P00022=2.006,1.622,-0.565,0.0000,0.0000,0.0000
///RCONF 0,0,0,0,0,0,0,0,0,0,0,0,0,0,0,0,0,0,0,0,0,0,0,0
P00023=-2.957,-4.083,2.762,0.0000,0.0000,0.0000
P00024=-1.466,-0.226,-0.419,0.0000,0.0000,0.0000
P00025=3.643,0.007,-2.585,0.0000,0.0000,0.0000
P00026=2.644,0.055,-2.583,0.0000,0.0000,0.0000
P00027=2.278,0.099,-4.210,0.0000,0.0000,0.0000
P00028=-1.778,-0.182,-2.050,0.0000,0.0000,0.0000
P00029=1.749,4.006,-0.261,0.0000,0.0000,0.0000
P00030=-0.014,-0.768,0.131,0.0000,0.0000,0.0000
P00031=-0.170,0.039,-0.647,0.0000,0.0000,0.0000
P00045=-8.836,-6.632,-1.438,0.0000,0.0000,0.0000
//INST
///DATE 2024/12/18 11:44
///ATTR SC,RW
///GROUP1 RB1,BS1
///GROUP2 ST1
NOP
'X2_99(90,0)
MOVJ C00000 BC00000 VJ=100.00  +MOVJ EC00000 VJ=100.00
MOVJ C00001 BC00001 VJ=100.00  +MOVJ EC00001 VJ=100.00
'Path S4826
SFTOF3D
MOVJ C00002 BC00002 VJ=100.00  +MOVJ EC00002 VJ=100.00
MOVL C00003 BC00003 V=800.0  +MOVJ EC00003 VJ=100.00
SMOVL C00004 BC00004 V=166.7  +MOVJ EC00004
SREFP 3 C00005 BC00005  +REFP EC00005
CALL JOB:SEARCH-R1-S13D
SET P031 P006
SFTON3D P031
SMOVL C00006 BC00006 V=166.7  +MOVJ EC00006
SREFP 3 C00007 BC00007  +REFP EC00007
CALL JOB:SEARCH-R1-S13D
SET P031 P006
SFTON3D P031
SMOVL C00008 BC00008 V=250.0  +MOVJ EC00008
SMOVL C00009 BC00009 V=250.0  +MOVJ EC00009
SREFP 3 C00010 BC00010  +REFP EC00010
CALL JOB:SEARCH-R1-S13D
SET P031 P006
SFTON3D P031
SMOVL C00011 BC00011 V=250.0  +MOVJ EC00011
MOVL C00012 BC00012 V=1000.0  +MOVJ EC00012 VJ=100.00
'EndPath S4826
MOVJ C00013 BC00013 VJ=100.00  +MOVJ EC00013 VJ=100.00
'Path S4869
SFTOF3D
MOVJ C00014 BC00014 VJ=100.00  +MOVJ EC00014 VJ=100.00
MOVL C00015 BC00015 V=800.0  +MOVJ EC00015 VJ=100.00
SMOVL C00016 BC00016 V=250.0  +MOVJ EC00016
SREFP 3 C00017 BC00017  +REFP EC00017
CALL JOB:SEARCH-R1-S13D
SET P030 P006
SFTON3D P030
SMOVL C00018 BC00018 V=166.7  +MOVJ EC00018
SMOVL C00019 BC00019 V=250.0  +MOVJ EC00019
SMOVL C00020 BC00020 V=250.0  +MOVJ EC00020
SMOVL C00021 BC00021 V=166.7  +MOVJ EC00021
SREFP 3 C00022 BC00022  +REFP EC00022
CALL JOB:SEARCH-R1-S13D
SET P030 P006
SFTON3D P030
SMOVL C00023 BC00023 V=250.0  +MOVJ EC00023
MOVL C00024 BC00024 V=1000.0  +MOVJ EC00024 VJ=100.00
'EndPath S4869
'Path S4870
SFTOF3D
MOVJ C00025 BC00025 VJ=100.00  +MOVJ EC00025 VJ=100.00
SMOVL C00026 BC00026 V=1000.0  +MOVJ EC00026
SMOVL C00027 BC00027 V=250.0  +MOVJ EC00027
SREFP 3 C00028 BC00028  +REFP EC00028
CALL JOB:SEARCH-R1-S13D
SET P029 P006
SFTON3D P029
SMOVL C00029 BC00029 V=250.0  +MOVJ EC00029
SMOVL C00030 BC00030 V=1000.0  +MOVJ EC00030
SMOVL C00031 BC00031 V=250.0  +MOVJ EC00031
SREFP 3 C00032 BC00032  +REFP EC00032
CALL JOB:SEARCH-R1-S13D
SET P029 P006
SFTON3D P029
SMOVL C00033 BC00033 V=250.0  +MOVJ EC00033
MOVL C00034 BC00034 V=1000.0  +MOVJ EC00034 VJ=100.00
'EndPath S4870
'Path S4823
SFTOF3D
MOVJ C00035 BC00035 VJ=100.00  +MOVJ EC00035 VJ=100.00
SMOVL C00036 BC00036 V=1000.0  +MOVJ EC00036
SMOVL C00037 BC00037 V=166.7  +MOVJ EC00037
SREFP 3 C00038 BC00038  +REFP EC00038
CALL JOB:SEARCH-R1-S13D
SET P028 P006
SFTON3D P028
SMOVL C00039 BC00039 V=250.0  +MOVJ EC00039
SMOVL C00040 BC00040 V=250.0  +MOVJ EC00040
SMOVL C00041 BC00041 V=250.0  +MOVJ EC00041
SREFP 3 C00042 BC00042  +REFP EC00042
CALL JOB:SEARCH-R1-S13D
SET P028 P006
SFTON3D P028
MOVL C00043 BC00043 V=1000.0  +MOVJ EC00043 VJ=100.00
SFTOF3D
SMOVL C00044 BC00044 V=1200.0  +MOVJ EC00044
SMOVL C00045 BC00045 V=1200.0  +MOVJ EC00045
SMOVL C00046 BC00046 V=166.7  +MOVJ EC00046
SREFP 3 C00047 BC00047  +REFP EC00047
CALL JOB:SEARCH-R1-S13D
SET P045 P006
SFTON3D P045
SMOVL C00048 BC00048 V=166.7  +MOVJ EC00048
SMOVL C00049 BC00049 V=800.0  +MOVJ EC00049
SMOVL C00050 BC00050 V=166.7  +MOVJ EC00050
SREFP 3 C00051 BC00051  +REFP EC00051
CALL JOB:SEARCH-R1-S13D
SET P045 P006
SFTON3D P045
SMOVL C00052 BC00052 V=166.7  +MOVJ EC00052
SMOVL C00053 BC00053 V=800.0  +MOVJ EC00053
SMOVL C00054 BC00054 V=800.0  +MOVJ EC00054
SMOVL C00055 BC00055 V=166.7  +MOVJ EC00055
SREFP 3 C00056 BC00056  +REFP EC00056
CALL JOB:SEARCH-R1-S13D
SET P045 P006
SFTON3D P045
SMOVL C00057 BC00057 V=250.0  +MOVJ EC00057
SMOVL C00058 BC00058 V=1200.0  +MOVJ EC00058
SFTOF3D
SMOVL C00059 BC00059 V=1200.0  +MOVJ EC00059
SMOVL C00060 BC00060 V=1200.0  +MOVJ EC00060
'EndPath S4823
'Path S4871
SFTOF3D
MOVJ C00061 BC00061 VJ=100.00  +MOVJ EC00061 VJ=100.00
MOVL C00062 BC00062 V=500.0  +MOVJ EC00062 VJ=100.00
SMOVL C00063 BC00063 V=166.7  +MOVJ EC00063
SREFP 3 C00064 BC00064  +REFP EC00064
CALL JOB:SEARCH-R1-S13D
SET P027 P006
SFTON3D P027
SMOVL C00065 BC00065 V=250.0  +MOVJ EC00065
SMOVL C00066 BC00066 V=166.7  +MOVJ EC00066
SREFP 3 C00067 BC00067  +REFP EC00067
CALL JOB:SEARCH-R1-S13D
SET P027 P006
SFTON3D P027
SMOVL C00068 BC00068 V=250.0  +MOVJ EC00068
MOVL C00069 BC00069 V=1000.0  +MOVJ EC00069 VJ=100.00
'EndPath S4871
'Path S4872
SFTOF3D
MOVJ C00070 BC00070 VJ=100.00  +MOVJ EC00070 VJ=100.00
MOVL C00071 BC00071 V=500.0  +MOVJ EC00071 VJ=100.00
SMOVL C00072 BC00072 V=166.7  +MOVJ EC00072
SREFP 3 C00073 BC00073  +REFP EC00073
CALL JOB:SEARCH-R1-S13D
SET P026 P006
SFTON3D P026
SMOVL C00074 BC00074 V=250.0  +MOVJ EC00074
SMOVL C00075 BC00075 V=166.7  +MOVJ EC00075
SREFP 3 C00076 BC00076  +REFP EC00076
CALL JOB:SEARCH-R1-S13D
SET P026 P006
SFTON3D P026
SMOVL C00077 BC00077 V=800.0  +MOVJ EC00077
MOVL C00078 BC00078 V=1000.0  +MOVJ EC00078 VJ=100.00
'EndPath S4872
'Path S4820
SFTOF3D
MOVJ C00079 BC00079 VJ=100.00  +MOVJ EC00079 VJ=100.00
MOVL C00080 BC00080 V=500.0  +MOVJ EC00080 VJ=100.00
SMOVL C00081 BC00081 V=166.7  +MOVJ EC00081
SREFP 3 C00082 BC00082  +REFP EC00082
CALL JOB:SEARCH-R1-S13D
SET P025 P006
SFTON3D P025
SMOVL C00083 BC00083 V=250.0  +MOVJ EC00083
SMOVL C00084 BC00084 V=166.7  +MOVJ EC00084
SREFP 3 C00085 BC00085  +REFP EC00085
CALL JOB:SEARCH-R1-S13D
SET P025 P006
SFTON3D P025
SMOVL C00086 BC00086 V=250.0  +MOVJ EC00086
MOVL C00087 BC00087 V=1000.0  +MOVJ EC00087 VJ=100.00
'EndPath S4820
MOVJ C00088 BC00088 VJ=100.00  +MOVJ EC00088 VJ=100.00
MOVJ C00089 BC00089 VJ=100.00  +MOVJ EC00089 VJ=100.00
'Path S4819 (for W4811)
SFTOF3D
MOVJ C00090 BC00090 VJ=100.00  +MOVJ EC00090 VJ=100.00
MOVL C00091 BC00091 V=666.7  +MOVJ EC00091 VJ=100.00
SMOVL C00092 BC00092 V=166.7  +MOVJ EC00092
SREFP 3 C00093 BC00093  +REFP EC00093
CALL JOB:SEARCH-R1-S13D
SET P024 P006
SFTON3D P024
SMOVL C00094 BC00094 V=166.7  +MOVJ EC00094
SREFP 3 C00095 BC00095  +REFP EC00095
CALL JOB:SEARCH-R1-S13D
SET P024 P006
SFTON3D P024
SMOVL C00096 BC00096 V=166.7  +MOVJ EC00096
MOVL C00097 BC00097 V=1000.0  +MOVJ EC00097 VJ=100.00
'EndPath S4819 (for W4811)
'Path S4818 (for W4811)
SFTOF3D
MOVJ C00098 BC00098 VJ=100.00  +MOVJ EC00098 VJ=100.00
MOVL C00099 BC00099 V=500.0  +MOVJ EC00099 VJ=100.00
SMOVL C00100 BC00100 V=166.7  +MOVJ EC00100
SREFP 3 C00101 BC00101  +REFP EC00101
CALL JOB:SEARCH-R1-S13D
SET P023 P006
SFTON3D P023
SMOVL C00102 BC00102 V=166.7  +MOVJ EC00102
SREFP 3 C00103 BC00103  +REFP EC00103
CALL JOB:SEARCH-R1-S13D
SET P023 P006
SFTON3D P023
SMOVL C00104 BC00104 V=166.7  +MOVJ EC00104
MOVL C00105 BC00105 V=1000.0  +MOVJ EC00105 VJ=100.00
'EndPath S4818 (for W4811)
MOVJ C00106 BC00106 VJ=100.00  +MOVJ EC00106 VJ=100.00
MOVJ C00107 BC00107 VJ=100.00  +MOVJ EC00107 VJ=100.00
MOVJ C00108 BC00108 VJ=100.00  +MOVJ EC00108 VJ=100.00
'Path S4816 (for W4808)
SFTOF3D
MOVJ C00109 BC00109 VJ=100.00  +MOVJ EC00109 VJ=100.00
MOVL C00110 BC00110 V=500.0  +MOVJ EC00110 VJ=100.00
SMOVL C00111 BC00111 V=166.7  +MOVJ EC00111
SREFP 3 C00112 BC00112  +REFP EC00112
CALL JOB:SEARCH-R1-S13D
SET P021 P006
SFTON3D P021
SMOVL C00113 BC00113 V=166.7  +MOVJ EC00113
SREFP 3 C00114 BC00114  +REFP EC00114
CALL JOB:SEARCH-R1-S13D
SET P021 P006
SFTON3D P021
SMOVL C00115 BC00115 V=166.7  +MOVJ EC00115
MOVL C00116 BC00116 V=1000.0  +MOVJ EC00116 VJ=100.00
'EndPath S4816 (for W4808)
MOVJ C00117 BC00117 VJ=100.00  +MOVJ EC00117 VJ=100.00
'Path S4817 (for W4808)
SFTOF3D
MOVJ C00118 BC00118 VJ=100.00  +MOVJ EC00118 VJ=100.00
MOVL C00119 BC00119 V=500.0  +MOVJ EC00119 VJ=100.00
SMOVL C00120 BC00120 V=166.7  +MOVJ EC00120
SREFP 3 C00121 BC00121  +REFP EC00121
CALL JOB:SEARCH-R1-S13D
SET P022 P006
SFTON3D P022
SMOVL C00122 BC00122 V=166.7  +MOVJ EC00122
SREFP 3 C00123 BC00123  +REFP EC00123
CALL JOB:SEARCH-R1-S13D
SET P022 P006
SFTON3D P022
SMOVL C00124 BC00124 V=166.7  +MOVJ EC00124
'EndPath S4817 (for W4808)
'Path W4808
SFTOF3D
SFTON3D P022
MOVJ C00125 BC00125 VJ=100.00  +MOVJ EC00125 VJ=100.00
SMOVL C00126 BC00126 V=800.0  +MOVJ EC00126
REFP 1 RB1 C00127 BC00127
REFP 1 RB1 C00128 BC00128
SMOVL C00129 BC00129 V=150.0 PL=0  +MOVJ EC00127
SWVON WEV#(100)
MACRO1 MJ#(0) ARGF21
ARCON
SMOVL C00130 BC00130 V=8.3  +MOVJ EC00128
SFTON3D P021
SMOVL C00131 BC00131 V=8.3  +MOVJ EC00129
SMOVL C00132 BC00132 V=8.3  +MOVJ EC00130
ARCOF
SWVOF
SMOVL C00133 BC00133 V=800.0  +MOVJ EC00131
SMOVL C00134 BC00134 V=1000.0  +MOVJ EC00132
SFTOF3D
'EndPath W4808
MOVJ C00135 BC00135 VJ=100.00  +MOVJ EC00133 VJ=100.00
MOVJ C00136 BC00136 VJ=100.00  +MOVJ EC00134 VJ=100.00
MOVJ C00137 BC00137 VJ=100.00  +MOVJ EC00135 VJ=100.00
MOVJ C00138 BC00138 VJ=100.00  +MOVJ EC00136 VJ=100.00
MOVJ C00139 BC00139 VJ=100.00  +MOVJ EC00137 VJ=100.00
'Path W4811
SFTOF3D
SFTON3D P024
MOVJ C00140 BC00140 VJ=100.00  +MOVJ EC00138 VJ=100.00
SMOVL C00141 BC00141 V=800.0  +MOVJ EC00139
REFP 1 RB1 C00142 BC00142
REFP 2 RB1 C00143 BC00143
SMOVL C00144 BC00144 V=150.0 PL=0  +MOVJ EC00140
MACRO1 MJ#(0) ARGF9
SWVON WEV#(100)
ARCON
SFTON3D P023
SMOVL C00145 BC00145 V=8.3  +MOVJ EC00141
ARCOF
SWVOF
SMOVL C00146 BC00146 V=800.0  +MOVJ EC00142
SMOVL C00147 BC00147 V=1000.0  +MOVJ EC00143
SFTOF3D
'EndPath W4811
'
MOVJ C00148 BC00148 VJ=100.00  +MOVJ EC00144 VJ=100.00
MOVJ C00149 BC00149 VJ=100.00  +MOVJ EC00145 VJ=100.00
MOVJ C00150 BC00150 VJ=100.00  +MOVJ EC00146 VJ=100.00
'Path W4873
SFTOF3D
SFTON3D P025
MOVJ C00151 BC00151 VJ=100.00  +MOVJ EC00147 VJ=100.00
SMOVL C00152 BC00152 V=800.0  +MOVJ EC00148
SMOVL C00153 BC00153 V=150.0 PL=0  +MOVJ EC00149
MACRO1 MJ#(0) ARGF14
ARCON
SMOVL C00154 BC00154 V=10.0  +MOVJ EC00150
SMOVL C00155 BC00155 V=10.8  +MOVJ EC00151
SFTON3D P026
SMOVL C00156 BC00156 V=10.8  +MOVJ EC00152
SFTON3D P027
SMOVL C00157 BC00157 V=10.8  +MOVJ EC00153
ARCOF
SMOVL C00158 BC00158 V=800.0  +MOVJ EC00154
SMOVL C00159 BC00159 V=1000.0  +MOVJ EC00155
SFTOF3D
COMM SFTON3D P025
COMM MOVJ C00160 BC00160 VJ=100.00  +MOVJ EC00156 VJ=100.00
COMM SMOVL C00161 BC00161 V=800.0  +MOVJ EC00157
COMM SMOVL C00162 BC00162 V=150.0 PL=0  +MOVJ EC00158
COMM MACRO1 MJ#(0) ARGF14
COMM ARCON
COMM SMOVL C00163 BC00163 V=10.8  +MOVJ EC00159
COMM ARCON
COMM SMOVL C00164 BC00164 V=10.0  +MOVJ EC00160
COMM ARCOF
COMM SMOVL C00165 BC00165 V=800.0  +MOVJ EC00161
COMM SMOVL C00166 BC00166 V=1000.0  +MOVJ EC00162
COMM SFTOF3D
COMM 'EndPath W4873
COMM 'Path W4874
COMM SFTOF3D
COMM SFTON3D P026
COMM MOVJ C00167 BC00167 VJ=100.00  +MOVJ EC00163 VJ=100.00
COMM SMOVL C00168 BC00168 V=800.0  +MOVJ EC00164
COMM SMOVL C00169 BC00169 V=150.0 PL=0  +MOVJ EC00165
COMM ARCON
COMM SMOVL C00170 BC00170 V=10.8  +MOVJ EC00166
COMM ARCOF
COMM SMOVL C00171 BC00171 V=800.0  +MOVJ EC00167
COMM SMOVL C00172 BC00172 V=1000.0  +MOVJ EC00168
COMM SFTOF3D
COMM 'EndPath W4874
COMM 'Path W4875
COMM SFTOF3D
COMM SFTON3D P027
COMM MOVJ C00173 BC00173 VJ=100.00  +MOVJ EC00169 VJ=100.00
COMM SMOVL C00174 BC00174 V=800.0  +MOVJ EC00170
COMM SMOVL C00175 BC00175 V=150.0 PL=0  +MOVJ EC00171
COMM ARCON
COMM SMOVL C00176 BC00176 V=10.8  +MOVJ EC00172
COMM ARCOF
COMM SMOVL C00177 BC00177 V=800.0  +MOVJ EC00173
COMM SMOVL C00178 BC00178 V=1000.0  +MOVJ EC00174
COMM SFTOF3D
'EndPath W4875
'Path W4876
SFTOF3D
SFTON3D P028
MOVJ C00179 BC00179 VJ=100.00  +MOVJ EC00175 VJ=100.00
SMOVL C00180 BC00180 V=800.0  +MOVJ EC00176
SMOVL C00181 BC00181 V=150.0 PL=0  +MOVJ EC00177
ARCON
SFTON3D P029
SMOVL C00182 BC00182 V=11.7  +MOVJ EC00178
SMOVL C00183 BC00183 V=11.7  +MOVJ EC00179
ARCOF
SMOVL C00184 BC00184 V=800.0  +MOVJ EC00180
SMOVL C00185 BC00185 V=1000.0  +MOVJ EC00181
SFTOF3D
'EndPath W4876
MOVJ C00186 BC00186 VJ=100.00  +MOVJ EC00182 VJ=100.00
MOVJ C00187 BC00187 VJ=100.00  +MOVJ EC00183 VJ=100.00
MOVJ C00188 BC00188 VJ=100.00  +MOVJ EC00184 VJ=100.00
'Path W4877
SFTOF3D
SFTON3D P030
MOVJ C00189 BC00189 VJ=100.00  +MOVJ EC00185 VJ=100.00
SMOVL C00190 BC00190 V=800.0  +MOVJ EC00186
SMOVL C00191 BC00191 V=150.0 PL=0  +MOVJ EC00187
ARCON
SMOVL C00192 BC00192 V=10.8  +MOVJ EC00188
SMOVL C00193 BC00193 V=10.8  +MOVJ EC00189
SMOVL C00194 BC00194 V=10.0  +MOVJ EC00190
ARCOF
SMOVL C00195 BC00195 V=800.0  +MOVJ EC00191
SMOVL C00196 BC00196 V=1000.0  +MOVJ EC00192
SFTOF3D
'EndPath W4877
MOVJ C00197 BC00197 VJ=100.00  +MOVJ EC00193 VJ=100.00
MOVJ C00198 BC00198 VJ=100.00  +MOVJ EC00194 VJ=100.00
'Path W4878
SFTOF3D
SFTON3D P031
MOVJ C00199 BC00199 VJ=100.00  +MOVJ EC00195 VJ=100.00
SMOVL C00200 BC00200 V=800.0  +MOVJ EC00196
MACRO1 MJ#(0) ARGF9
SMOVL C00201 BC00201 V=150.0 PL=0  +MOVJ EC00197
ARCON
SMOVL C00202 BC00202 V=10.0 PL=0  +MOVJ EC00198
ARCON
SWVON WEV#(101)
SMOVL C00203 BC00203 V=8.3  +MOVJ EC00199
SMOVL C00204 BC00204 V=8.3  +MOVJ EC00200
SWVOF
SFTON3D P030
MACRO1 MJ#(0) ARGF14
SMOVL C00205 BC00205 V=10.0  +MOVJ EC00201
ARCOF
SMOVL C00206 BC00206 V=800.0  +MOVJ EC00202
SMOVL C00207 BC00207 V=1000.0  +MOVJ EC00203
SFTOF3D
'EndPath W4878
MOVJ C00208 BC00208 VJ=100.00  +MOVJ EC00204 VJ=100.00
MOVJ C00209 BC00209 VJ=100.00  +MOVJ EC00205 VJ=100.00
MOVJ C00210 BC00210 VJ=100.00  +MOVJ EC00206 VJ=100.00
SFTON3D P045
MACRO1 MJ#(0) ARGF6
SMOVL C00211 BC00211 V=166.7  +MOVJ EC00207
ARCON
SMOVL C00212 BC00212 V=10.0  +MOVJ EC00208
ARCOF
SMOVL C00213 BC00213 V=166.7  +MOVJ EC00209
SMOVL C00214 BC00214 V=166.7  +MOVJ EC00210
SMOVL C00215 BC00215 V=166.7  +MOVJ EC00211
ARCON
SMOVL C00216 BC00216 V=11.7  +MOVJ EC00212
ARCOF
SMOVL C00217 BC00217 V=250.0  +MOVJ EC00213
MOVJ C00218 BC00218 VJ=100.00  +MOVJ EC00214 VJ=100.00
MOVJ C00219 BC00219 VJ=100.00  +MOVJ EC00215 VJ=100.00
MOVJ C00220 BC00220 VJ=100.00  +MOVJ EC00216 VJ=100.00
SMOVL C00221 BC00221 V=166.7  +MOVJ EC00217
SMOVL C00222 BC00222 V=11.7  +MOVJ EC00218
ARCOF
SMOVL C00223 BC00223 V=800.0  +MOVJ EC00219
SFTOF3D
MOVJ C00224 BC00224 VJ=100.00  +MOVJ EC00220 VJ=100.00
MOVJ C00225 BC00225 VJ=100.00  +MOVJ EC00221 VJ=100.00
MOVJ C00226 BC00226 VJ=100.00  +MOVJ EC00222 VJ=100.00
MOVJ C00227 BC00227 VJ=100.00  +MOVJ EC00223 VJ=100.00
MOVJ C00228 BC00228 VJ=100.00  +MOVJ EC00224 VJ=100.00
CALL JOB:CLEAN-R1_KM_NEW
'
'
'
'
'
'
'Path S4829
SFTOF3D
MOVJ C00229 BC00229 VJ=100.00  +MOVJ EC00225 VJ=100.00
MOVJ C00230 BC00230 VJ=100.00  +MOVJ EC00226 VJ=100.00
MOVL C00231 BC00231 V=666.7  +MOVJ EC00227 VJ=100.00
SMOVL C00232 BC00232 V=166.7  +MOVJ EC00228
SREFP 3 C00233 BC00233  +REFP EC00229
CALL JOB:SEARCH-R1-S13D
SET P031 P006
SFTON3D P031
SMOVL C00234 BC00234 V=166.7  +MOVJ EC00230
SREFP 3 C00235 BC00235  +REFP EC00231
CALL JOB:SEARCH-R1-S13D
SET P031 P006
SFTON3D P031
SMOVL C00236 BC00236 V=166.7  +MOVJ EC00232
SMOVL C00237 BC00237 V=666.7  +MOVJ EC00233
SMOVL C00238 BC00238 V=166.7  +MOVJ EC00234
SREFP 3 C00239 BC00239  +REFP EC00235
CALL JOB:SEARCH-R1-S13D
SET P031 P006
SFTON3D P031
SMOVL C00240 BC00240 V=166.7  +MOVJ EC00236
'EndPath S4829
MOVJ C00241 BC00241 VJ=100.00  +MOVJ EC00237 VJ=100.00
'Path S4830
SFTOF3D
MOVJ C00242 BC00242 VJ=100.00  +MOVJ EC00238 VJ=100.00
SMOVL C00243 BC00243 V=666.7  +MOVJ EC00239
SMOVL C00244 BC00244 V=166.7  +MOVJ EC00240
SREFP 3 C00245 BC00245  +REFP EC00241
CALL JOB:SEARCH-R1-S13D
SET P030 P006
SFTON3D P030
SMOVL C00246 BC00246 V=166.7  +MOVJ EC00242
SMOVL C00247 BC00247 V=666.7  +MOVJ EC00243
SMOVL C00248 BC00248 V=166.7  +MOVJ EC00244
SREFP 3 C00249 BC00249  +REFP EC00245
CALL JOB:SEARCH-R1-S13D
SET P030 P006
SFTON3D P030
SMOVL C00250 BC00250 V=250.0  +MOVJ EC00246
MOVL C00251 BC00251 V=1000.0  +MOVJ EC00247 VJ=100.00
'EndPath S4830
'Path S4831
SFTOF3D
MOVJ C00252 BC00252 VJ=100.00  +MOVJ EC00248 VJ=100.00
SMOVL C00253 BC00253 V=666.7  +MOVJ EC00249
SMOVL C00254 BC00254 V=166.7  +MOVJ EC00250
SREFP 3 C00255 BC00255  +REFP EC00251
CALL JOB:SEARCH-R1-S13D
SET P029 P006
SFTON3D P029
SMOVL C00256 BC00256 V=166.7  +MOVJ EC00252
SMOVL C00257 BC00257 V=666.7  +MOVJ EC00253
SMOVL C00258 BC00258 V=166.7  +MOVJ EC00254
SREFP 3 C00259 BC00259  +REFP EC00255
CALL JOB:SEARCH-R1-S13D
SET P029 P006
SFTON3D P029
SMOVL C00260 BC00260 V=250.0  +MOVJ EC00256
MOVL C00261 BC00261 V=1000.0  +MOVJ EC00257 VJ=100.00
'EndPath S4831
'Path S4832
SFTOF3D
SMOVL C00262 BC00262 V=1200.0  +MOVJ EC00258
SMOVL C00263 BC00263 V=1000.0  +MOVJ EC00259
SMOVL C00264 BC00264 V=166.7  +MOVJ EC00260
SREFP 3 C00265 BC00265  +REFP EC00261
CALL JOB:SEARCH-R1-S13D
SET P045 P006
SFTON3D P045
SMOVL C00266 BC00266 V=166.7  +MOVJ EC00262
SMOVL C00267 BC00267 V=333.3  +MOVJ EC00263
SMOVL C00268 BC00268 V=166.7  +MOVJ EC00264
SREFP 3 C00269 BC00269  +REFP EC00265
CALL JOB:SEARCH-R1-S13D
SET P045 P006
SFTON3D P045
SMOVL C00270 BC00270 V=166.7  +MOVJ EC00266
SMOVL C00271 BC00271 V=800.0  +MOVJ EC00267
SMOVL C00272 BC00272 V=166.7  +MOVJ EC00268
SREFP 3 C00273 BC00273  +REFP EC00269
CALL JOB:SEARCH-R1-S13D
SET P045 P006
SFTON3D P045
SMOVL C00274 BC00274 V=166.7  +MOVJ EC00270
SFTOF3D
SMOVL C00275 BC00275 V=1000.0  +MOVJ EC00271
SMOVL C00276 BC00276 V=1200.0  +MOVJ EC00272
SMOVL C00277 BC00277 V=666.7  +MOVJ EC00273
SMOVL C00278 BC00278 V=166.7  +MOVJ EC00274
SREFP 3 C00279 BC00279  +REFP EC00275
CALL JOB:SEARCH-R1-S13D
SET P028 P006
SFTON3D P028
SMOVL C00280 BC00280 V=166.7  +MOVJ EC00276
SMOVL C00281 BC00281 V=666.7  +MOVJ EC00277
SMOVL C00282 BC00282 V=166.7  +MOVJ EC00278
SREFP 3 C00283 BC00283  +REFP EC00279
CALL JOB:SEARCH-R1-S13D
SET P028 P006
SFTON3D P028
SMOVL C00284 BC00284 V=166.7  +MOVJ EC00280
MOVL C00285 BC00285 V=1000.0  +MOVJ EC00281 VJ=100.00
'EndPath S4832
MOVJ C00286 BC00286 VJ=100.00  +MOVJ EC00282 VJ=100.00
'Path S4833
SFTOF3D
MOVJ C00287 BC00287 VJ=100.00  +MOVJ EC00283 VJ=100.00
MOVL C00288 BC00288 V=666.7  +MOVJ EC00284 VJ=100.00
SMOVL C00289 BC00289 V=166.7  +MOVJ EC00285
SREFP 3 C00290 BC00290  +REFP EC00286
CALL JOB:SEARCH-R1-S13D
SET P027 P006
SFTON3D P027
SMOVL C00291 BC00291 V=166.7  +MOVJ EC00287
SMOVL C00292 BC00292 V=166.7  +MOVJ EC00288
SREFP 3 C00293 BC00293  +REFP EC00289
CALL JOB:SEARCH-R1-S13D
SET P027 P006
SFTON3D P027
SMOVL C00294 BC00294 V=166.7  +MOVJ EC00290
MOVL C00295 BC00295 V=1000.0  +MOVJ EC00291 VJ=100.00
'EndPath S4833
'Path S4834
SFTOF3D
MOVJ C00296 BC00296 VJ=100.00  +MOVJ EC00292 VJ=100.00
MOVL C00297 BC00297 V=666.7  +MOVJ EC00293 VJ=100.00
SMOVL C00298 BC00298 V=166.7  +MOVJ EC00294
SREFP 3 C00299 BC00299  +REFP EC00295
CALL JOB:SEARCH-R1-S13D
SET P026 P006
SFTON3D P026
SMOVL C00300 BC00300 V=166.7  +MOVJ EC00296
SMOVL C00301 BC00301 V=166.7  +MOVJ EC00297
SREFP 3 C00302 BC00302  +REFP EC00298
CALL JOB:SEARCH-R1-S13D
SET P026 P006
SFTON3D P026
SMOVL C00303 BC00303 V=166.7  +MOVJ EC00299
'EndPath S4834
'Path S4835
SFTOF3D
MOVJ C00304 BC00304 VJ=100.00  +MOVJ EC00300 VJ=100.00
MOVL C00305 BC00305 V=666.7  +MOVJ EC00301 VJ=100.00
SMOVL C00306 BC00306 V=166.7  +MOVJ EC00302
SREFP 3 C00307 BC00307  +REFP EC00303
CALL JOB:SEARCH-R1-S13D
SET P025 P006
SFTON3D P025
SMOVL C00308 BC00308 V=166.7  +MOVJ EC00304
SMOVL C00309 BC00309 V=166.7  +MOVJ EC00305
SREFP 3 C00310 BC00310  +REFP EC00306
CALL JOB:SEARCH-R1-S13D
SET P025 P006
SFTON3D P025
SMOVL C00311 BC00311 V=166.7  +MOVJ EC00307
MOVL C00312 BC00312 V=1000.0  +MOVJ EC00308 VJ=100.00
'EndPath S4835
MOVJ C00313 BC00313 VJ=100.00  +MOVJ EC00309 VJ=100.00
MOVJ C00314 BC00314 VJ=100.00  +MOVJ EC00310 VJ=100.00
'Path S4836 (for W4841)
SFTOF3D
MOVJ C00315 BC00315 VJ=100.00  +MOVJ EC00311 VJ=100.00
MOVL C00316 BC00316 V=666.7  +MOVJ EC00312 VJ=100.00
SMOVL C00317 BC00317 V=166.7  +MOVJ EC00313
SREFP 3 C00318 BC00318  +REFP EC00314
CALL JOB:SEARCH-R1-S13D
SET P024 P006
SFTON3D P024
SMOVL C00319 BC00319 V=166.7  +MOVJ EC00315
SREFP 3 C00320 BC00320  +REFP EC00316
CALL JOB:SEARCH-R1-S13D
SET P024 P006
SFTON3D P024
SMOVL C00321 BC00321 V=166.7  +MOVJ EC00317
MOVL C00322 BC00322 V=1000.0  +MOVJ EC00318 VJ=100.00
'EndPath S4836 (for W4841)
'Path S4837 (for W4841)
SFTOF3D
MOVJ C00323 BC00323 VJ=100.00  +MOVJ EC00319 VJ=100.00
MOVL C00324 BC00324 V=666.7  +MOVJ EC00320 VJ=100.00
SMOVL C00325 BC00325 V=166.7  +MOVJ EC00321
SREFP 3 C00326 BC00326  +REFP EC00322
CALL JOB:SEARCH-R1-S13D
SET P023 P006
SFTON3D P023
SMOVL C00327 BC00327 V=166.7  +MOVJ EC00323
SREFP 3 C00328 BC00328  +REFP EC00324
CALL JOB:SEARCH-R1-S13D
SET P023 P006
SFTON3D P023
SMOVL C00329 BC00329 V=166.7  +MOVJ EC00325
MOVL C00330 BC00330 V=1000.0  +MOVJ EC00326 VJ=100.00
'EndPath S4837 (for W4841)
MOVJ C00331 BC00331 VJ=100.00  +MOVJ EC00327 VJ=100.00
MOVJ C00332 BC00332 VJ=100.00  +MOVJ EC00328 VJ=100.00
MOVJ C00333 BC00333 VJ=100.00  +MOVJ EC00329 VJ=100.00
MOVJ C00334 BC00334 VJ=100.00  +MOVJ EC00330 VJ=100.00
'Path S4838 (for W4840)
SFTOF3D
MOVJ C00335 BC00335 VJ=100.00  +MOVJ EC00331 VJ=100.00
MOVL C00336 BC00336 V=666.7  +MOVJ EC00332 VJ=100.00
SMOVL C00337 BC00337 V=166.7  +MOVJ EC00333
SREFP 3 C00338 BC00338  +REFP EC00334
CALL JOB:SEARCH-R1-S13D
SET P021 P006
SFTON3D P021
SMOVL C00339 BC00339 V=166.7  +MOVJ EC00335
SREFP 3 C00340 BC00340  +REFP EC00336
CALL JOB:SEARCH-R1-S13D
SET P021 P006
SFTON3D P021
SMOVL C00341 BC00341 V=166.7  +MOVJ EC00337
MOVL C00342 BC00342 V=1000.0  +MOVJ EC00338 VJ=100.00
'EndPath S4838 (for W4840)
MOVJ C00343 BC00343 VJ=100.00  +MOVJ EC00339 VJ=100.00
'Path S4839 (for W4840)
SFTOF3D
MOVJ C00344 BC00344 VJ=100.00  +MOVJ EC00340 VJ=100.00
MOVL C00345 BC00345 V=666.7  +MOVJ EC00341 VJ=100.00
SMOVL C00346 BC00346 V=166.7  +MOVJ EC00342
SREFP 3 C00347 BC00347  +REFP EC00343
CALL JOB:SEARCH-R1-S13D
SET P022 P006
SFTON3D P022
SMOVL C00348 BC00348 V=166.7  +MOVJ EC00344
SREFP 3 C00349 BC00349  +REFP EC00345
CALL JOB:SEARCH-R1-S13D
SET P022 P006
SFTON3D P022
SMOVL C00350 BC00350 V=166.7  +MOVJ EC00346
'EndPath S4839 (for W4840)
'Path W4840
SFTOF3D
SFTON3D P022
SMOVL C00351 BC00351 V=800.0  +MOVJ EC00347
SREFP 1 C00352 BC00352  +REFP EC00348
SREFP 2 C00353 BC00353  +REFP EC00349
SMOVL C00354 BC00354 V=150.0 PL=0  +MOVJ EC00350
MACRO1 MJ#(0) ARGF21
ARCON
SWVON WEV#(100)
SFTON3D P021
SMOVL C00355 BC00355 V=8.3  +MOVJ EC00351
ARCOF
SWVOF
SMOVL C00356 BC00356 V=800.0  +MOVJ EC00352
SMOVL C00357 BC00357 V=1000.0  +MOVJ EC00353
SFTOF3D
'EndPath W4840
MOVJ C00358 BC00358 VJ=100.00  +MOVJ EC00354 VJ=100.00
MOVJ C00359 BC00359 VJ=100.00  +MOVJ EC00355 VJ=100.00
MOVJ C00360 BC00360 VJ=100.00  +MOVJ EC00356 VJ=100.00
MOVJ C00361 BC00361 VJ=100.00  +MOVJ EC00357 VJ=100.00
'Path W4841
SFTOF3D
SFTON3D P024
MOVJ C00362 BC00362 VJ=100.00  +MOVJ EC00358 VJ=100.00
SMOVL C00363 BC00363 V=800.0  +MOVJ EC00359
SMOVL C00364 BC00364 V=150.0 PL=0  +MOVJ EC00360
ARCON
SWVON WEV#(100)
SFTON3D P023
SMOVL C00365 BC00365 V=8.3  +MOVJ EC00361
ARCOF
SWVOF
SMOVL C00366 BC00366 V=800.0  +MOVJ EC00362
SMOVL C00367 BC00367 V=1000.0  +MOVJ EC00363
SFTOF3D
'EndPath W4841
'
MOVJ C00368 BC00368 VJ=100.00  +MOVJ EC00364 VJ=100.00
'Path W4842
SFTOF3D
SFTON3D P025
MOVJ C00369 BC00369 VJ=100.00  +MOVJ EC00365 VJ=100.00
SMOVL C00370 BC00370 V=800.0  +MOVJ EC00366
SMOVL C00371 BC00371 V=150.0 PL=0  +MOVJ EC00367
MACRO1 MJ#(0) ARGF14
ARCON
SMOVL C00372 BC00372 V=10.8  +MOVJ EC00368
SFTON3D P026
SMOVL C00373 BC00373 V=10.8  +MOVJ EC00369
SFTON3D P027
SMOVL C00374 BC00374 V=10.8  +MOVJ EC00370
ARCOF
SMOVL C00375 BC00375 V=800.0  +MOVJ EC00371
SMOVL C00376 BC00376 V=1000.0  +MOVJ EC00372
SFTOF3D
COMM SFTON3D P025
COMM MOVJ C00377 BC00377 VJ=100.00  +MOVJ EC00373 VJ=100.00
COMM SMOVL C00378 BC00378 V=800.0  +MOVJ EC00374
COMM SMOVL C00379 BC00379 V=150.0 PL=0  +MOVJ EC00375
COMM MACRO1 MJ#(0) ARGF9
COMM ARCON
COMM SMOVL C00380 BC00380 V=12.5  +MOVJ EC00376
COMM ARCOF
COMM SMOVL C00381 BC00381 V=800.0  +MOVJ EC00377
COMM SMOVL C00382 BC00382 V=1000.0  +MOVJ EC00378
COMM SFTOF3D
COMM 'EndPath W4842
COMM 'Path W4843
COMM SFTOF3D
COMM SFTON3D P026
COMM MOVJ C00383 BC00383 VJ=100.00  +MOVJ EC00379 VJ=100.00
COMM SMOVL C00384 BC00384 V=800.0  +MOVJ EC00380
COMM SMOVL C00385 BC00385 V=150.0 PL=0  +MOVJ EC00381
COMM ARCON
COMM SMOVL C00386 BC00386 V=12.5  +MOVJ EC00382
COMM ARCOF
COMM SMOVL C00387 BC00387 V=800.0  +MOVJ EC00383
COMM SMOVL C00388 BC00388 V=1000.0  +MOVJ EC00384
COMM SFTOF3D
COMM 'EndPath W4843
COMM 'Path W4844
COMM SFTOF3D
COMM SFTON3D P027
COMM MOVJ C00389 BC00389 VJ=100.00  +MOVJ EC00385 VJ=100.00
COMM SMOVL C00390 BC00390 V=800.0  +MOVJ EC00386
COMM SMOVL C00391 BC00391 V=150.0 PL=0  +MOVJ EC00387
COMM ARCON
COMM SMOVL C00392 BC00392 V=12.5  +MOVJ EC00388
COMM ARCOF
COMM SMOVL C00393 BC00393 V=800.0  +MOVJ EC00389
COMM SMOVL C00394 BC00394 V=1000.0  +MOVJ EC00390
COMM SFTOF3D
'EndPath W4844
'Path W4845
SFTOF3D
SFTON3D P028
MOVJ C00395 BC00395 VJ=100.00  +MOVJ EC00391 VJ=100.00
SMOVL C00396 BC00396 V=800.0  +MOVJ EC00392
SMOVL C00397 BC00397 V=150.0 PL=0  +MOVJ EC00393
MACRO1 MJ#(0) ARGF14
ARCON
SFTON3D P029
SMOVL C00398 BC00398 V=10.0  +MOVJ EC00394
SMOVL C00399 BC00399 V=10.0  +MOVJ EC00395
ARCOF
SMOVL C00400 BC00400 V=800.0  +MOVJ EC00396
SMOVL C00401 BC00401 V=1000.0  +MOVJ EC00397
SFTOF3D
'EndPath W4845
MOVJ C00402 BC00402 VJ=100.00  +MOVJ EC00398 VJ=100.00
MOVJ C00403 BC00403 VJ=100.00  +MOVJ EC00399 VJ=100.00
MOVJ C00404 BC00404 VJ=100.00  +MOVJ EC00400 VJ=100.00
'Path W4846
SFTOF3D
SFTON3D P030
MOVJ C00405 BC00405 VJ=100.00  +MOVJ EC00401 VJ=100.00
SMOVL C00406 BC00406 V=800.0  +MOVJ EC00402
SMOVL C00407 BC00407 V=150.0 PL=0  +MOVJ EC00403
ARCON
SMOVL C00408 BC00408 V=10.8  +MOVJ EC00404
SMOVL C00409 BC00409 V=10.8  +MOVJ EC00405
SMOVL C00410 BC00410 V=12.5  +MOVJ EC00406
SMOVL C00411 BC00411 V=12.5  +MOVJ EC00407
ARCOF
SMOVL C00412 BC00412 V=800.0  +MOVJ EC00408
SMOVL C00413 BC00413 V=1000.0  +MOVJ EC00409
SFTOF3D
'EndPath W4846
MOVJ C00414 BC00414 VJ=100.00  +MOVJ EC00410 VJ=100.00
MOVJ C00415 BC00415 VJ=100.00  +MOVJ EC00411 VJ=100.00
'Path W4847
SFTOF3D
SFTON3D P031
MOVJ C00416 BC00416 VJ=100.00  +MOVJ EC00412 VJ=100.00
SMOVL C00417 BC00417 V=800.0  +MOVJ EC00413
SMOVL C00418 BC00418 V=150.0 PL=0  +MOVJ EC00414
MACRO1 MJ#(0) ARGF9
ARCON
SWVON WEV#(101)
SMOVL C00419 BC00419 V=10.0 PL=0  +MOVJ EC00415
SMOVL C00420 BC00420 V=8.3  +MOVJ EC00416
SMOVL C00421 BC00421 V=8.3  +MOVJ EC00417
SWVOF
SFTON3D P030
SMOVL C00422 BC00422 V=10.0  +MOVJ EC00418
ARCOF
SMOVL C00423 BC00423 V=800.0  +MOVJ EC00419
SMOVL C00424 BC00424 V=1000.0  +MOVJ EC00420
SFTOF3D
'EndPath W4847
MOVJ C00425 BC00425 VJ=100.00  +MOVJ EC00421 VJ=100.00
MOVJ C00426 BC00426 VJ=100.00  +MOVJ EC00422 VJ=100.00
MACRO1 MJ#(0) ARGF6
MOVJ C00427 BC00427 VJ=80.00  +MOVJ EC00423 VJ=80.00
MOVJ C00428 BC00428 VJ=100.00  +MOVJ EC00424 VJ=100.00
SFTOF3D
END
